Fanuc KAREL source: kx00021.KL

-- PROVISIONAL review KL for V1013-1; original PC SHA256 e615e17a03ad453a0f15783d98712fa48473d1b20aae57ad2c33e5d2e6d289da
-- Incomplete behavior may be omitted. Consult companion uncertainty JSON. Do not deploy.
PROGRAM KX00021
%NOLOCKGROUP
BEGIN
  -- UNRESOLVED_PC offsets 5-25; opcodes 2E,22,9D,33,2E,33,35
  -- UNRESOLVED_PC offsets 30-51; opcodes 22,9D,33,2E,33,34,23
  -- UNRESOLVED_PC offsets 56-60; opcodes 7F
END KX00021
